TYPE ST_TransferMoldErrors_OLD :
STRUCT
	HydraulicCilinder			: ST_HydraulicErrorsAnalog;

	Error1: BOOL;
	Error2: BOOL;

END_STRUCT
END_TYPE

(* stored: Version 1.1.0.1, ProductVersion 3.1.4020.12
   DUT ST_TransferMoldErrors_OLD: Id {a320b9f0-e122-4b37-97b4-1ff6db1e57e7} *)
